{attribute addProperty BoxType "EK1122-0000-0018"}
{attribute addProperty Id "Beckhoff_EPP7xxxsub_EK1100EK1100_179A0949162A_0001_EPP7041_1002_0016EPP7041_5614098424030A_0002_EPP7041_1002_0017EPP7041_5614098424030A_0003_EPP7041_1002_0023EPP7041_E93814AC24030A_0004_EPP7041_3002_0016EPP7041_E93814AC24030A_0005_EPP7041_3002_0017EPP7041_E93814AC24030A_0006_EPP7041_3002_0018EPP7041_E93814AC24030A_0007_EPP7041_3002_0023EPP7041_E93814AC24030A_0008_EPP7342_0002_0016EPP7342_014E044838448A_0009_EPP7342_0002_0017EPP7342_014E044838448"}
{attribute addProperty CRC "2510970711"}
{attribute addProperty SizeInBites "2464"}
{attribute addProperty SizeInBytes "308"}
TYPE Beckhoff_EPP7xxxEK1122_95AA5F57 EXTENDS EK1122_179A0949 :
STRUCT
	{attribute addProperty Name "Beckhoff_EPP7xxxsub_EK1100"}
	Beckhoff_EPP7xxxsub_EK1100 : EK1100_179A0949;
	{attribute addProperty Name "A_0001_EPP7041_1002_0016"}
	A_0001_EPP7041_1002_0016 : EPP7041_56140984;
	{attribute addProperty Name "A_0002_EPP7041_1002_0017"}
	A_0002_EPP7041_1002_0017 : EPP7041_56140984;
	{attribute addProperty Name "A_0003_EPP7041_1002_0023"}
	A_0003_EPP7041_1002_0023 : EPP7041_E93814AC;
	{attribute addProperty Name "A_0004_EPP7041_3002_0016"}
	A_0004_EPP7041_3002_0016 : EPP7041_E93814AC;
	{attribute addProperty Name "A_0005_EPP7041_3002_0017"}
	A_0005_EPP7041_3002_0017 : EPP7041_E93814AC;
	{attribute addProperty Name "A_0006_EPP7041_3002_0018"}
	A_0006_EPP7041_3002_0018 : EPP7041_E93814AC;
	{attribute addProperty Name "A_0007_EPP7041_3002_0023"}
	A_0007_EPP7041_3002_0023 : EPP7041_E93814AC;
	{attribute addProperty Name "A_0008_EPP7342_0002_0016"}
	A_0008_EPP7342_0002_0016 : EPP7342_014E0448;
	{attribute addProperty Name "A_0009_EPP7342_0002_0017"}
	A_0009_EPP7342_0002_0017 : EPP7342_014E0448;
END_STRUCT
END_TYPE

(* stored: Version 1.2.0.0, ProductVersion 3.1.4024.9
   DUT Beckhoff_EPP7xxxEK1122_95AA5F57: Id {7d11bfb8-4ba3-4015-b08d-0f35a85ca23f} *)
